FUNCTION_BLOCK FB_MatrixElementSum_Test EXTENDS FB_TestSuite
VAR_INPUT
END_VAR
VAR_OUTPUT
END_VAR
VAR
END_VAR

WhenDifferentExpectError();
WhenmatchingExpectResult();

METHOD PRIVATE WhenDifferentExpectError
VAR_INPUT
END_VAR
VAR
	M1 : DynamicMatrix;
	M2 : DynamicMatrix;
	M3 : DynamicMatrix;
	Result : BOOL;
END_VAR
TEST('WhenDifferentExpectError');

// @TEST-RUN
M1.InitMagicSquare(3);
M2.InitMagicSquare(5);
Result := M3.AsElementSum(M1,M2);

// @TEST-ASSERT
AssertFalse(Result,'Main function call was unexpectedly successful');

TEST_FINISHED();
END_METHOD

METHOD PRIVATE WhenMatchingExpectResult
VAR_INPUT
END_VAR
VAR
	M1 : DynamicMatrix;
	M2 : DynamicMatrix;
	M3 : DynamicMatrix;
	Result : BOOL;
END_VAR
TEST('WhenMatchingExpectResult');

// @TEST-RUN
M1.InitMagicSquare(3);
M2.InitMagicSquare(3);
Result := M3.AsElementSum(M1,M2);
M1.Scale(2);

// @TEST-ASSERT
AssertTrue(Result,'Main function call was not successful');
AssertTrue(M3.IsEqual(M1),'Data was successfully added');

TEST_FINISHED();
END_METHOD

END_FUNCTION_BLOCK

(* stored: Version 1.1.0.1, ProductVersion 3.1.4024.9
   POU FB_MatrixElementSum_Test: Id {4dcbf96e-83e7-0942-1466-313401dfc7f7}, SpecialFunc None
   Method WhenDifferentExpectError: Id {7c8500e5-8b06-049b-26ef-8c68b2165305}
   Method WhenMatchingExpectResult: Id {4704fc92-c368-0aa0-2102-7dfaed302d6f} *)
